// TIA Portal V20 export
TYPE "typeSequenceControlNodeJobInterface"
// stored: Namespace Unit1.Em2
   STRUCT
      commands { ExternalWritable := 'False'} : "Unit1.Em2.typeSequenceControlNodeJobInterfaceCommands";
      monitoring { ExternalWritable := 'False'} : "Unit1.Em2.typeSequenceControlNodeJobInterfaceMonitoring";
   END_STRUCT;
END_TYPE
